{attribute 'qualified_only'}
{attribute 'strict'}
{attribute 'to_string'}
TYPE E_LIST_CTRL :
(
  LIST_CTRL_INVALID,
	LIST_CTRL_NULL,
  LIST_CTRL_INIT      := 10,
  LIST_CTRL_GET_HEAD  := 20,
  LIST_CTRL_GET_TAIL  := 30,
  LIST_CTRL_ADD_HEAD  := 40,
  LIST_CTRL_ADD_TAIL  := 50,
  LIST_CTRL_DEL_HEAD  := 60,
  LIST_CTRL_DEL_TAIL  := 70
)UINT;
END_TYPE

(* stored: Version 1.1.0.1
   DUT E_LIST_CTRL: Id {0b879881-7244-497f-a8e0-825d0822a259} *)
